// TIA Portal project "Sorting Boxes using Factory IO Simulation" (V17)

(* hardware
DEVICE "S7-1200 station_1"  S7-1200 Station
   slot 0: "Rack_0"  S7-1200 Rack  Rack  V1.0
   slot 1: "PLC_1"  CPU 1215C AC/DC/Rly  6ES7 215-1BG40-0XB0  V4.5
*)

// ===== PLC "PLC_1"  CPU 1215C AC/DC/Rly =====

VAR_GLOBAL   // PLC tag table "Default tag table"
   "Height_sensor_1" AT %I0.0 : Bool;
   "Height_sensor_2" AT %I0.1 : Bool;
   "Height_sensor_3" AT %I0.2 : Bool;
   "Load" AT %I0.3 : Bool;
   "Left Entry" AT %I0.4 : Bool;
   "Right Entry" AT %I0.5 : Bool;
   "Start_Button_1" AT %I1.0 : Bool;
   "Reset_Button_1" AT %I1.1 : Bool;
   "Feed Conveyor" AT %Q0.0 : Bool;
   "Load Sensor" AT %Q0.1 : Bool;
   "Unload" AT %Q0.2 : Bool;
   "Chain_Transfer_Left" AT %Q0.3 : Bool;
   "Chain_Transfer_Right" AT %Q0.4 : Bool;
   "Left_Conveyor" AT %Q0.5 : Bool;
   "Right_Conveyor" AT %Q0.6 : Bool;
   "Reset Light" AT %Q0.7 : Bool;
   "Start Light" AT %Q1.0 : Bool;
   "Remover 1" AT %Q1.1 : Bool;
   "Remover 2" AT %Q1.2 : Bool;
   "Emitter" AT %Q1.3 : Bool;
   "Tag_1" AT %M0.0 : Bool;
   "Tag_2" AT %M0.1 : Bool;
   "Tag_3" AT %MD1 : Time;
   "Tag_4" AT %M0.5 : Bool;
   "Tag_5" AT %M0.2 : Bool;
   "Tag_6" AT %M0.7 : Bool;
   "Tag_7" AT %M2.0 : Bool;
   "right counter" AT %QW34 : Int;
   "Tag_8" AT %M2.1 : Bool;
   "Left counter" AT %QW30 : Int;
   "Tag_9" AT %M10.0 : Bool;
END_VAR

// folder: System blocks/Program resources

DATA_BLOCK "IEC_Timer_0_DB"   // DB1
{ S7_Optimized_Access := 'TRUE' }
AUTHOR : Simatic
FAMILY : IEC
NAME : IEC_TMR
VERSION : 1.0
// stored: InstanceOfName IEC_TIMER
"IEC_TIMER"
BEGIN
END_DATA_BLOCK

DATA_BLOCK "IEC_Timer_0_DB_1"   // DB2
{ S7_Optimized_Access := 'TRUE' }
AUTHOR : Simatic
FAMILY : IEC
NAME : IEC_TMR
VERSION : 1.0
// stored: InstanceOfName IEC_TIMER
"IEC_TIMER"
BEGIN
END_DATA_BLOCK

DATA_BLOCK "IEC_Counter_0_DB"   // DB3
{ S7_Optimized_Access := 'TRUE' }
AUTHOR : Simatic
FAMILY : IEC
NAME : CNTR
VERSION : 1.0
// stored: InstanceOfName IEC_COUNTER
"IEC_COUNTER"
BEGIN
END_DATA_BLOCK

DATA_BLOCK "IEC_Counter_0_DB_1"   // DB4
{ S7_Optimized_Access := 'TRUE' }
AUTHOR : Simatic
FAMILY : IEC
NAME : CNTR
VERSION : 1.0
// stored: InstanceOfName IEC_COUNTER
"IEC_COUNTER"
BEGIN
END_DATA_BLOCK

DATA_BLOCK "IEC_Timer_0_DB_2"   // DB5
{ S7_Optimized_Access := 'TRUE' }
AUTHOR : Simatic
FAMILY : IEC
NAME : IEC_TMR
VERSION : 1.0
// stored: InstanceOfName IEC_TIMER
"IEC_TIMER"
BEGIN
END_DATA_BLOCK

// folder: (top level)

FUNCTION "MHJ-PLC-Lab-Function-S71200" : Void   // FC9000, SCL
{ S7_Optimized_Access := 'TRUE' }
VERSION : 0.1
   VAR_TEMP
      rdTimeReturn : Int;
      outputTime : DTL;
      SyncVal : Byte;
      forVal : Int;
      forVal_2 : Int;
      Value : Byte;
   END_VAR
   VAR CONSTANT
      CompVal : Byte := 16#34;
      Value_01 : Byte := 16#11;
      Value_01_DW : DWord := 16#A165_D992;
      Value_02_DW : DWord := 16#58BE_4401;
   END_VAR
BEGIN

   #Value:=PEEK(area := 16#82,
        dbNumber := 0,
        byteOffset := 511);
   #Value := #Value + 1;

   POKE(area := 16#82,
        dbNumber := 0,
        byteOffset := 511,
        value := #Value);

   POKE(area:=16#81,
        dbNumber:=0,
        byteOffset:=1016,
        value:=#Value_01_DW);
   POKE(area := 16#81,
        dbNumber := 0,
        byteOffset := 1020,
        value := #Value_02_DW);

   POKE(area := 16#81,
        dbNumber := 0,
        byteOffset := 511,
        value := B#16#00);

   FOR #forVal := 0 TO 120 DO
       FOR #forVal_2:=0 TO 10 DO
           #rdTimeReturn:=RD_SYS_T(#outputTime);
           #rdTimeReturn := WR_SYS_T(#outputTime);
           #rdTimeReturn := RD_SYS_T(#outputTime);
           #rdTimeReturn := WR_SYS_T(#outputTime);
       END_FOR;
       #SyncVal:= PEEK(area := 16#81,
                      dbNumber := 0,
                      byteOffset := 511);
       IF #SyncVal = #CompVal THEN
          GOTO M_1;
       END_IF;
   END_FOR;
   RETURN;

   M_1:
   POKE(area := 16#81,
        dbNumber := 0,
        byteOffset := 511,
        value := B#16#0);
END_FUNCTION

ORGANIZATION_BLOCK "Main"   // OB1, LAD, ProgramCycle
TITLE = "Main Program Sweep (Cycle)"
{ S7_Optimized_Access := 'TRUE' }
VERSION : 0.1
   VAR_INPUT
      Initial_Call : Bool;   // Initial call of this OB
      Remanence : Bool;   // =True, if remanent data are available
   END_VAR
   VAR_TEMP   // added for the SCL form of the ladder/FBD networks
      _w1 : Bool;
   END_VAR
BEGIN

REGION Network 1
   // Factory IO Communication Configuration
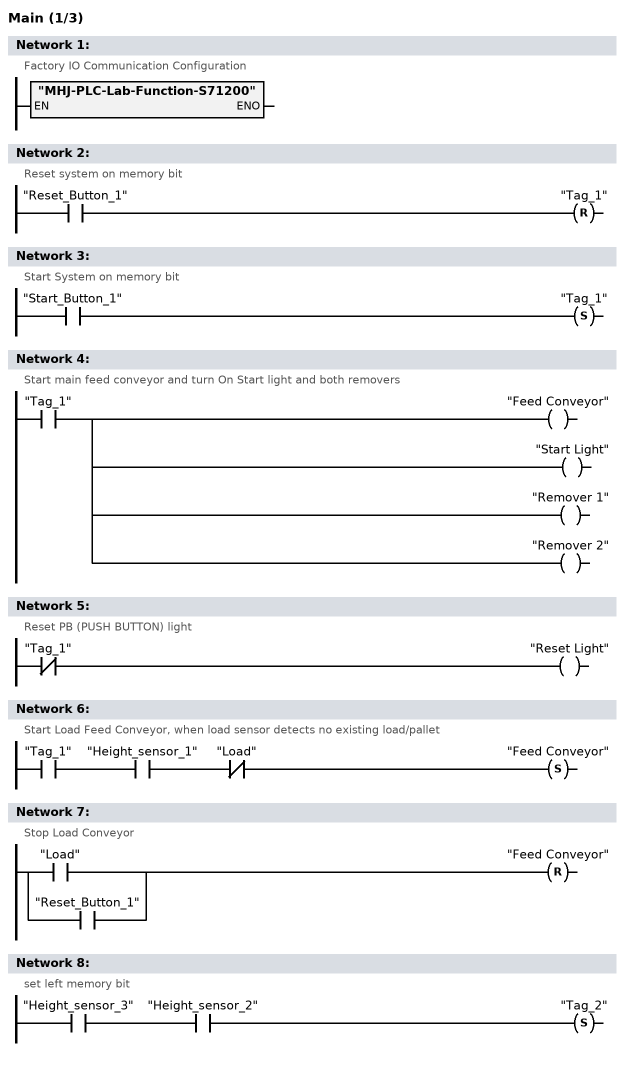
   RUNG wire#powerrail
      "MHJ-PLC-Lab-Function-S71200"()
   END_RUNG
   // the same network as SCL:
   "MHJ-PLC-Lab-Function-S71200"();
END_REGION

REGION Network 2
   // Reset system on memory bit
   RUNG wire#powerrail
      Contact( "Reset_Button_1" )
      R_Coil( "Tag_1" )
   END_RUNG
   // the same network as SCL:
   IF "Reset_Button_1" THEN "Tag_1" := FALSE; END_IF;
END_REGION

REGION Network 3
   // Start System on memory bit
   RUNG wire#powerrail
      Contact( "Start_Button_1" )
      S_Coil( "Tag_1" )
   END_RUNG
   // the same network as SCL:
   IF "Start_Button_1" THEN "Tag_1" := TRUE; END_IF;
END_REGION

REGION Network 4
   // Start main feed conveyor and turn On Start light and both removers
   RUNG wire#powerrail
      Contact( "Tag_1" )
      wire#w1
      Coil( "Feed Conveyor" )
   END_RUNG
   RUNG wire#w1
      Coil( "Start Light" )
   END_RUNG
   RUNG wire#w1
      Coil( "Remover 1" )
   END_RUNG
   RUNG wire#w1
      Coil( "Remover 2" )
   END_RUNG
   // the same network as SCL:
   "Feed Conveyor" := "Tag_1";
   "Start Light" := "Tag_1";
   "Remover 1" := "Tag_1";
   "Remover 2" := "Tag_1";
END_REGION

REGION Network 5
   // Reset PB (PUSH BUTTON) light
   RUNG wire#powerrail
      I_Contact( "Tag_1" )
      Coil( "Reset Light" )
   END_RUNG
   // the same network as SCL:
   "Reset Light" := NOT "Tag_1";
END_REGION

REGION Network 6
   // Start Load Feed Conveyor, when load sensor detects no existing load/pallet
   RUNG wire#powerrail
      Contact( "Tag_1" )
      Contact( "Height_sensor_1" )
      I_Contact( "Load" )
      S_Coil( "Feed Conveyor" )
   END_RUNG
   // the same network as SCL:
   IF "Tag_1" AND "Height_sensor_1" AND NOT "Load" THEN "Feed Conveyor" := TRUE; END_IF;
END_REGION

REGION Network 7
   // Stop Load Conveyor
   RUNG wire#powerrail
      Contact( "Load" )
      wire#w1
      R_Coil( "Feed Conveyor" )
   END_RUNG
   RUNG wire#powerrail
      Contact( "Reset_Button_1" )
   END_RUNG wire#w1
   // the same network as SCL:
   IF "Load" OR "Reset_Button_1" THEN "Feed Conveyor" := FALSE; END_IF;
END_REGION

REGION Network 8
   // set left memory bit
   RUNG wire#powerrail
      Contact( "Height_sensor_3" )
      Contact( "Height_sensor_2" )
      S_Coil( "Tag_2" )
   END_RUNG
   // the same network as SCL:
   IF "Height_sensor_3" AND "Height_sensor_2" THEN "Tag_2" := TRUE; END_IF;
END_REGION

REGION Network 9
   // Turn ON chain left transfer & left conveyor
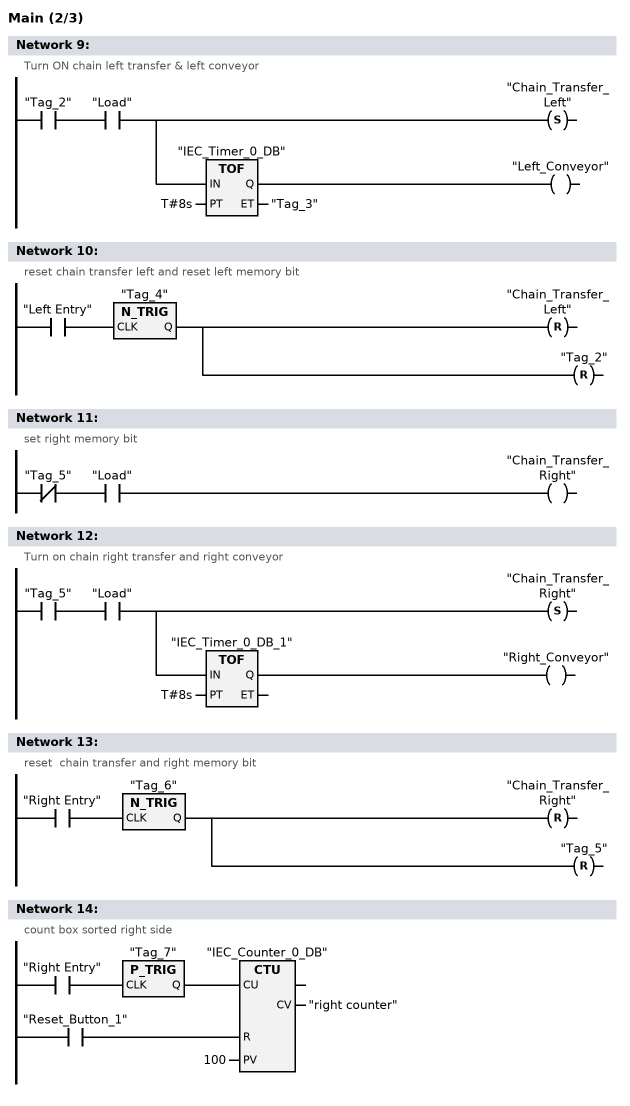
   #_w1 := "Tag_2" AND "Load";
   IF #_w1 THEN "Chain_Transfer_Left" := TRUE; END_IF;
   "IEC_Timer_0_DB".TOF(IN := #_w1, PT := T#8s, ET => "Tag_3");
   "Left_Conveyor" := "IEC_Timer_0_DB".Q;
END_REGION

REGION Network 10
   // reset chain transfer left and reset left memory bit
   RUNG wire#powerrail
      Contact( "Left Entry" )
      N_Trig( "Tag_4" )
      wire#w1
      R_Coil( "Chain_Transfer_Left" )
   END_RUNG
   RUNG wire#w1
      R_Coil( "Tag_2" )
   END_RUNG
   // the same network as SCL:
   #_w1 := NOT "Left Entry" AND "Tag_4";   // falling edge
   "Tag_4" := "Left Entry";
   IF #_w1 THEN
       "Chain_Transfer_Left" := FALSE;
       "Tag_2" := FALSE;
   END_IF;
END_REGION

REGION Network 11
   // set right memory bit
   RUNG wire#powerrail
      I_Contact( "Tag_5" )
      Contact( "Load" )
      Coil( "Chain_Transfer_Right" )
   END_RUNG
   // the same network as SCL:
   "Chain_Transfer_Right" := NOT "Tag_5" AND "Load";
END_REGION

REGION Network 12
   // Turn on chain right transfer and right conveyor
   #_w1 := "Tag_5" AND "Load";
   IF #_w1 THEN "Chain_Transfer_Right" := TRUE; END_IF;
   "IEC_Timer_0_DB_1".TOF(IN := #_w1, PT := T#8s);
   "Right_Conveyor" := "IEC_Timer_0_DB_1".Q;
END_REGION

REGION Network 13
   // reset  chain transfer and right memory bit
   RUNG wire#powerrail
      Contact( "Right Entry" )
      N_Trig( "Tag_6" )
      wire#w1
      R_Coil( "Chain_Transfer_Right" )
   END_RUNG
   RUNG wire#w1
      R_Coil( "Tag_5" )
   END_RUNG
   // the same network as SCL:
   #_w1 := NOT "Right Entry" AND "Tag_6";   // falling edge
   "Tag_6" := "Right Entry";
   IF #_w1 THEN
       "Chain_Transfer_Right" := FALSE;
       "Tag_5" := FALSE;
   END_IF;
END_REGION

REGION Network 14
   // count box sorted right side
   #_w1 := "Right Entry" AND NOT "Tag_7";   // rising edge
   "Tag_7" := "Right Entry";
   "IEC_Counter_0_DB".CTU(CU := #_w1, R := "Reset_Button_1", PV := 100, CV => "right counter");
END_REGION

REGION Network 15
   // count box sorted left side
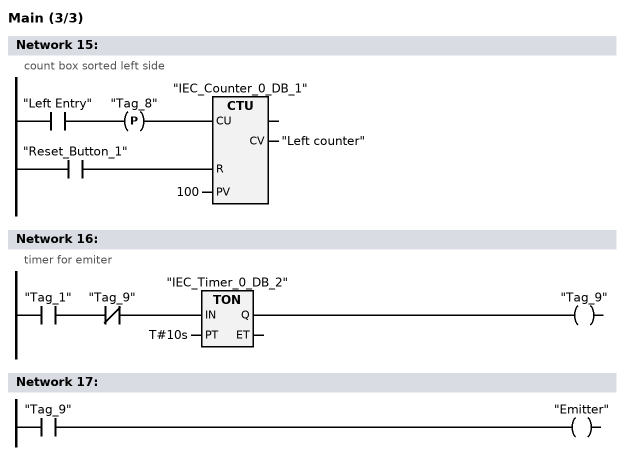
   #_w1 := "Left Entry" AND NOT "Tag_8";   // rising edge
   "Tag_8" := "Left Entry";
   "IEC_Counter_0_DB_1".CTU(CU := #_w1, R := "Reset_Button_1", PV := 100, CV => "Left counter");
END_REGION

REGION Network 16
   // timer for emiter
   "IEC_Timer_0_DB_2".TON(IN := "Tag_1" AND NOT "Tag_9", PT := T#10s);
   "Tag_9" := "IEC_Timer_0_DB_2".Q;
END_REGION

REGION Network 17
   RUNG wire#powerrail
      Contact( "Tag_9" )
      Coil( "Emitter" )
   END_RUNG
   // the same network as SCL:
   "Emitter" := "Tag_9";
END_REGION
END_ORGANIZATION_BLOCK